// TIA Portal V18 export
DATA_BLOCK "Alarm_DB"   // DB36
{ S7_Optimized_Access := 'FALSE' }
VERSION : 0.1
// stored: AutoNumber true, DBAccessibleFromOPCUA true, IsOnlyStoredInLoadMemory false, IsWriteProtectedInAS false
   VAR
      input : Struct
         alarm : Array[0..95] of Bool;   // Connect the alarm inputs according to the alarm list
         ack : Array[0..95] of Bool;
      END_STRUCT;
      output : Struct
         alarm_reg : Array[0..95] of Bool;
      END_STRUCT;
      i : Int;
      alarmhmi : Bool;
      alarmRegister1 : Word;
      alarmRegister2 : Word;
      alarmRegister3 : Word;
      alarmRegister4 : Word;
      alarmRegister5 : Word;
      reset : Array[0..95] of Bool;
   END_VAR
BEGIN
   // input.alarm[0] : reg1 bit 8
   // input.alarm[1] : reg1 bit 9
   // input.alarm[2] : reg1 bit 10
   // input.alarm[3] : reg1 bit 11
   // input.alarm[4] : reg1 bit 12
   // input.alarm[5] : reg1 bit 13
   // input.alarm[6] : reg1 bit 14
   // input.alarm[7] : reg1 bit 15
   // input.alarm[8] : reg1 bit 0
   // input.alarm[9] : reg1 bit 1
   // input.alarm[10] : reg1 bit 2
   // input.alarm[11] : reg1 bit 3
   // input.alarm[12] : reg1 bit 4
   // input.alarm[13] : reg1 bit 5
   // input.alarm[14] : reg1 bit 6
   // input.alarm[15] : reg1 bit 0
   // input.alarm[16] : reg2 bit 8
   // input.alarm[17] : reg2 bit 9
   // input.alarm[18] : reg2 bit 10
   // input.alarm[19] : reg2 bit 11
   // input.alarm[20] : reg2 bit 12
   // input.alarm[21] : reg2 bit 13
   // input.alarm[22] : reg2 bit 14
   // input.alarm[23] : reg2 bit 15
   // input.alarm[24] : reg2 bit 7
   // input.alarm[25] : reg2 bit 6
   // input.alarm[26] : reg2 bit 5
   // input.alarm[27] : reg2 bit 4
   // input.alarm[28] : reg2 bit 3
   // input.alarm[29] : reg2 bit 2
   // input.alarm[30] : reg2 bit 1
   // input.alarm[31] : reg2 bit 0
   // input.alarm[32] : reg3 bit 8
   // input.alarm[33] : reg3 bit 9
   // input.alarm[34] : reg3 bit 10
   // input.alarm[35] : reg3 bit 11
   // input.alarm[36] : reg3 bit 12
   // input.alarm[37] : reg3 bit 13
   // input.alarm[38] : reg3 bit 14
   // input.alarm[39] : reg3 bit 15
   // input.alarm[40] : reg3 bit 7
   // input.alarm[41] : reg3 bit 6
   // input.alarm[42] : reg3 bit 5
   // input.alarm[43] : reg3 bit 4
   // input.alarm[44] : reg3 bit 3
   // input.alarm[45] : reg3 bit 2
   // input.alarm[46] : reg3 bit 1
   // input.alarm[47] : reg3 bit 0
   // input.alarm[48] : reg4 bit 8
   // input.alarm[49] : reg4 bit 9
   // input.alarm[50] : reg4 bit 10
   // input.alarm[51] : reg4 bit 11
   // input.alarm[52] : reg4 bit 12
   // input.alarm[53] : reg4 bit 13
   // input.alarm[54] : reg4 bit 14
   // input.alarm[55] : reg4 bit 15
   // input.alarm[56] : reg4 bit 7
   // input.alarm[57] : reg4 bit 6
   // input.alarm[58] : reg4 bit 5
   // input.alarm[59] : reg4 bit 4
   // input.alarm[60] : reg4 bit 3
   // input.alarm[61] : reg4 bit 2
   // input.alarm[62] : reg4 bit 1
   // input.alarm[63] : reg4 bit 0
   // input.alarm[64] : reg5 bit 8
   // input.alarm[65] : reg5 bit 9
   // input.alarm[66] : reg5 bit 10
   // input.alarm[67] : reg5 bit 11
   // input.alarm[68] : reg5 bit 12
   // input.alarm[69] : reg5 bit 13
   // input.alarm[70] : reg5 bit 14
   // input.alarm[71] : reg5 bit 15
   // input.alarm[72] : reg5 bit 7
   // input.alarm[73] : reg5 bit 6
   // input.alarm[74] : reg5 bit 5
   // input.alarm[75] : reg5 bit 4
   // input.alarm[76] : reg5 bit 3
   // input.alarm[77] : reg5 bit 2
   // input.alarm[78] : reg5 bit 1
   // input.alarm[79] : reg5 bit 0
END_DATA_BLOCK
